	FUNCTION_BLOCK FB 141
	TITLE =G041M AERATION AIR STEEPING 5
	//COPYRIGHT:    (C) 2009  BUHLER AG, CH-9240 UZWIL, SWITZERLAND
	//
	//PRODUCT:      WinCoS_BIW01_09
	//
	//TITLE:        AERATION AIR STEEPING 5
	//                Machine group control
	//                Maschinengruppensteuerung
	//
	//--------------------------------------------------------------------------------
	//
	//IDENT:        AUTHOR:             DEPT:                              DATE:
	//
	//P01_FB141.1.0 K.Renz              CSB41                              13.Jan.2010
	//             1st Release
	//
	//--------------------------------------------------------------------------------
	//
	//PURPOSE:
	//
	//MANUAL :
	//
	//RESTRICTIONS:
	//
	//--------------------------------------------------------------------------------
	AUTHOR  : KR
	FAMILY  : USW
	VERSION : 9.9


	VAR
	  Gr       : FB10;	//Standard interface to group
	  InOutValue1    : DINT; //Data for user
	  InOutValue2    : DINT; //Data for user
	  OutWayConflict : BOOL;	//Data for user
	  OutSelectionOk : BOOL;	//Data for user
	  CmdNewValue : BOOL;	//Data for user
	  CmdNewJob   : BOOL;	//Data for user
	  OutCodeOK   : BOOL;	//Data for user
	  InEndOfJob  : BOOL ;	//Data for user
	  staWayOk      : BOOL ;	//Data for user
	  EdgeStartRelease : BOOL ;	//Data for user
	  USW8  : BOOL;	//Data for user
	  USW9 : BOOL;	//Data for user
	  USW10: BOOL;	//Data for user
	  USW11: BOOL;	//Data for user
	  USW12: BOOL;	//Data for user
	  USW13: BOOL;	//Data for user
	  USW14: BOOL;	//Data for user
	  USW15: BOOL;	//Data for user
	     #A_1115_QXV_BZS41_42 : FB13;   // VLS
	     #A_1115_MXZ45_BZS47_48 : FB13;   // VLS
	END_VAR
	VAR_TEMP
	   tmpEnable		: BOOL;
	   tmpFlag  		: BOOL;
	   tmpCmdNext		: BOOL;
	   tmpLocal  		: BOOL;
	   tmpAspOk  		: BOOL;
	   tmpHWStop 		: BOOL;
	   tmpInstanzDBNo       : INT ;
	END_VAR
	BEGIN
	NETWORK
	TITLE =
	NETWORK
	TITLE =Read command from group control
	//Parameter
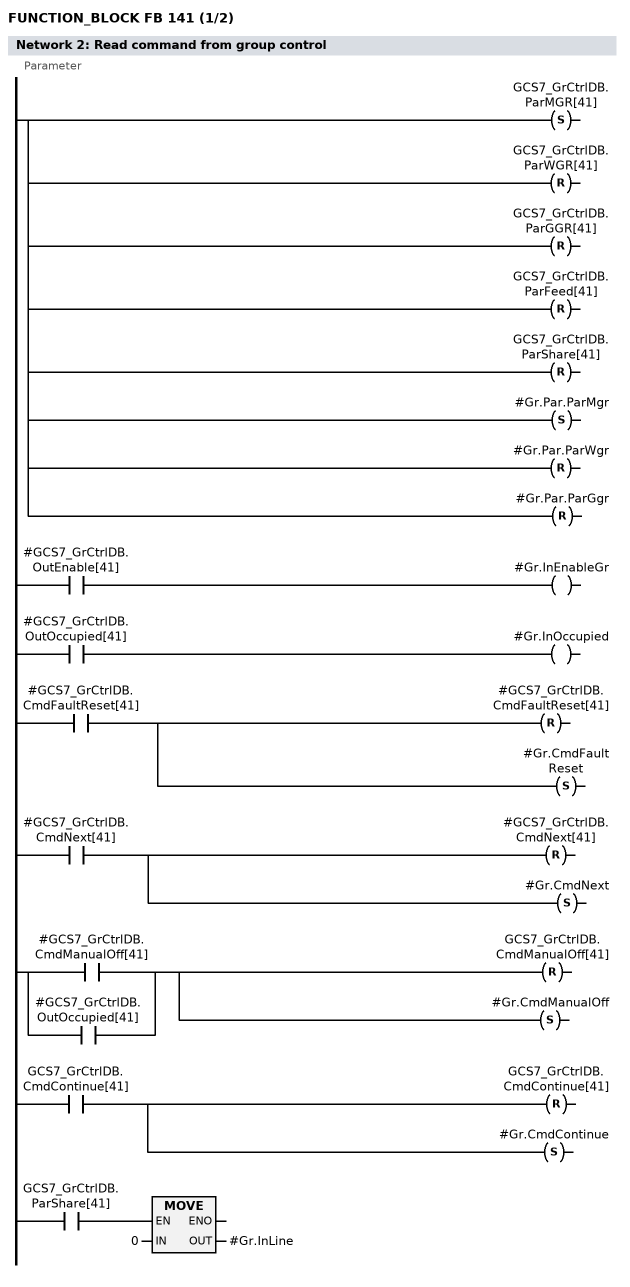
	      SET;
	      S   GCS7_GrCtrlDB.ParMGR[41];
	      R   GCS7_GrCtrlDB.ParWGR[41];
	      R   GCS7_GrCtrlDB.ParGGR[41];
	      R   GCS7_GrCtrlDB.ParFeed[41];
	      R   GCS7_GrCtrlDB.ParShare[41];
	      S   #Gr.Par.ParMgr;
	      R   #Gr.Par.ParWgr;
	      R   #Gr.Par.ParGgr;
	//Command
	      U   #GCS7_GrCtrlDB.OutEnable[41];
	      =   #Gr.InEnableGr;
	      U   #GCS7_GrCtrlDB.OutOccupied[41];
	      =   #Gr.InOccupied;
	      U   #GCS7_GrCtrlDB.CmdFaultReset[41];
	      R   #GCS7_GrCtrlDB.CmdFaultReset[41];
	      S   #Gr.CmdFaultReset;
	      U  #GCS7_GrCtrlDB.CmdNext[41];
	      R   #GCS7_GrCtrlDB.CmdNext[41];
	      S   #Gr.CmdNext;
	      U   #GCS7_GrCtrlDB.CmdManualOff[41];
	      O   #GCS7_GrCtrlDB.OutOccupied[41];
	      R   GCS7_GrCtrlDB.CmdManualOff[41];
	      S   #Gr.CmdManualOff;
	      U  GCS7_GrCtrlDB.CmdContinue[41];
	      R   GCS7_GrCtrlDB.CmdContinue[41];
	      S   #Gr.CmdContinue;
	//Init Line Number
	      U   GCS7_GrCtrlDB.ParShare[41];
	      SPBN WE00;
	      L     0;
	      T     #Gr.InLine;
	WE00: NOP   0;
	NETWORK
	TITLE =Call Methode Control
	// 1. Handle Interface PCControl
	// 2. Prepare mode --> ModePassive,ModeActive,ModeIdling
	// 3. Reset global flags of the group
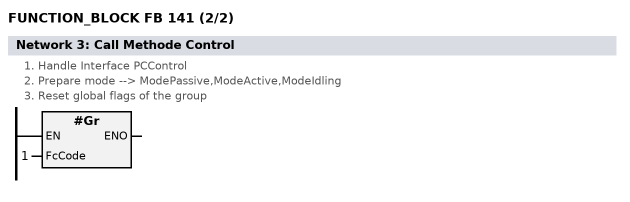
	      CALL #Gr (
	           FcCode                   := 1);
	NETWORK
	TITLE =Restart Idling Time
		L  #Gr.Par.ParIdling;
		L  2;
		>=I;
		SPB IdTm;
		T  #Gr.Par.ParIdling;
	IdTm:   NOP 0;
	      CLR;
	      S    #Gr.CmdRestartIdling;
	NETWORK
	TITLE =Prepare global flags
	NETWORK
	TITLE =Set Pattern (Target position)
	NETWORK
	TITLE =Interlocking WayOk
	//
	NETWORK
	TITLE =Interlocking Autostart
		CLR;
		R   #Gr.OutAutostart;
	NETWORK
	TITLE =Interlocking Enable
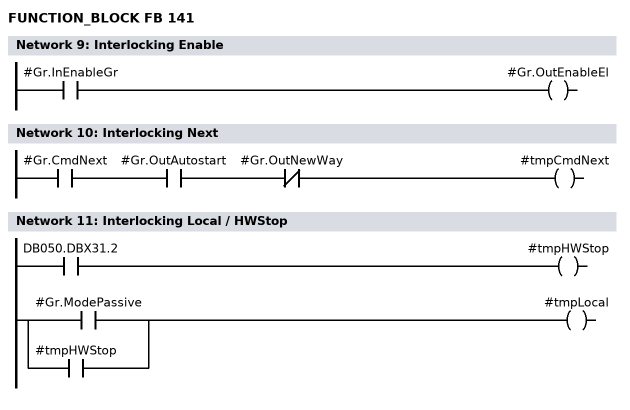
	      U     #Gr.InEnableGr;
	      =     #Gr.OutEnableEl;

	NETWORK
	TITLE =Interlocking Next
	      U     #Gr.CmdNext;
	      U     #Gr.OutAutostart;
	      UN    #Gr.OutNewWay;
	      =    #tmpCmdNext;

	NETWORK
	TITLE =Interlocking Local / HWStop
	      U    DB050.DBX31.2;
	      =    #tmpHWStop;

	      U    #Gr.ModePassive;
	      O    #tmpHWStop;
	      =    #tmpLocal;

	NETWORK
	TITLE =Interlocking Start Warning
	      NOP 0;
	//- Restart after fault --
	      U     #Gr.CmdFaultReset;
	      U     #Gr.VarFault;
	      S       "SYS_StartWarningDB".Area[1].CmdResetStartWarning;
	//- Run Timer --
	      AUF "G041M";
	      CALL  FB100 , DB100(
	       InModeHigher :=FALSE,
	       InArea     :=1,
	       InEnable   :=#Gr.OutEnableEl,
	       InLocal    :=#tmpLocal,
	       InStarted  :=#Gr.VarStarted,
	       InCmdNext  :=#tmpCmdNext,
	       OutCmdNext :=#tmpCmdNext,
	       OutStartwarning:=#Gr.VarStartWarning);
	//- Store Startwarning done  --
	//- Reset Autostart --
	      U     "SYS_StartWarningDB".TmpArea.OutStartReleaseRunningL;
	      FN    #EdgeStartRelease;
	      U     #Gr.VarFault;
	      R     #Gr.OutAutostart;
	NETWORK
	TITLE ==A-1115-QXV/BZS41/42 : AERATION AIR RING ST 5
	NOP 0;
	//-InLocal---
	      U     #tmpLocal;
	      =     #A_1115_QXV_BZS41_42.InLocal;
	//
	//-Interlocking---
	         =     #A_1115_QXV_BZS41_42.InEnableHN;
	         NOT;
	         =     #A_1115_QXV_BZS41_42.InEnableLN;
	//
	         SET;
	         S     #A_1115_QXV_BZS41_42.CmdNext;
	//
	      U     #Gr.OutSeqStop;
	      =     #A_1115_QXV_BZS41_42.InSeqStop;
	//
	//-Read inputs---
	      U     E 033.0;
	      =     #A_1115_QXV_BZS41_42.InpLN;
	      U     E 033.1;
	      =     #A_1115_QXV_BZS41_42.InpHN;
	      U   DB050.DBX31.2;
	      =     #A_1115_QXV_BZS41_42.InHWStop;
	       U     PLC_DPInfo.Master[1].SlavesError[6];
	       =       #A_1115_QXV_BZS41_42.InDPFault;
	//
	//-Set Parameters---
	//
	//-Call object control---
	      CALL  #A_1115_QXV_BZS41_42;
	//
	//-Write outputs---
	      U     #A_1115_QXV_BZS41_42.OutpHN;
	      =     A 033.1;
	NETWORK
	TITLE ==A-1115-MXZ45/BZS47/48 : AERATION AIR TUBE ST 5
	NOP 0;
	//-InLocal---
	      U     #tmpLocal;
	      =     #A_1115_MXZ45_BZS47_48.InLocal;
	//
	//-Interlocking---
	      	      U(;
	      U     #A_1115_QXV_BZS41_42.InEnableLN;
	      U     #A_1115_QXV_BZS41_42.StLN;
	      O;
	      U     #A_1115_QXV_BZS41_42.InEnableHN;
	      U     #A_1115_QXV_BZS41_42.StHN;
	      );
	         =     #A_1115_MXZ45_BZS47_48.InEnableHN;
	         NOT;
	         =     #A_1115_MXZ45_BZS47_48.InEnableLN;
	//
	         SET;
	         S     #A_1115_MXZ45_BZS47_48.CmdNext;
	//
	      U     #Gr.OutSeqStop;
	      =     #A_1115_MXZ45_BZS47_48.InSeqStop;
	//
	//-Read inputs---
	      U     E 066.2;
	      =     #A_1115_MXZ45_BZS47_48.InpLN;
	      U     E 066.3;
	      =     #A_1115_MXZ45_BZS47_48.InpHN;
	      X     A 065.1;
	      X     E 066.1;
	      O;
	      X     A 065.0;
	      X     E 066.0;
	      =     #A_1115_MXZ45_BZS47_48.InpFaultDev;
	      U   DB050.DBX31.2;
	      =     #A_1115_MXZ45_BZS47_48.InHWStop;
	       U     PLC_DPInfo.Master[1].SlavesError[10];
	       =       #A_1115_MXZ45_BZS47_48.InDPFault;
	//
	//-Set Parameters---
	//
	//-Call object control---
	      CALL  #A_1115_MXZ45_BZS47_48;
	//
	//-Write outputs---
	      U     #A_1115_MXZ45_BZS47_48.OutpLN;
	      =     A 065.1;
	      U     #A_1115_MXZ45_BZS47_48.OutpHN;
	      =     A 065.0;
	NETWORK
	TITLE =Test Fault
	      U     #A_1115_QXV_BZS41_42.StFault;
	      O     #A_1115_MXZ45_BZS47_48.StFault;
	      =     #Gr.VarFault;
	NETWORK
	TITLE =Test Warning
	      CLR;
	      =     #Gr.OutWarning;
	NETWORK
	TITLE =Test Stopped
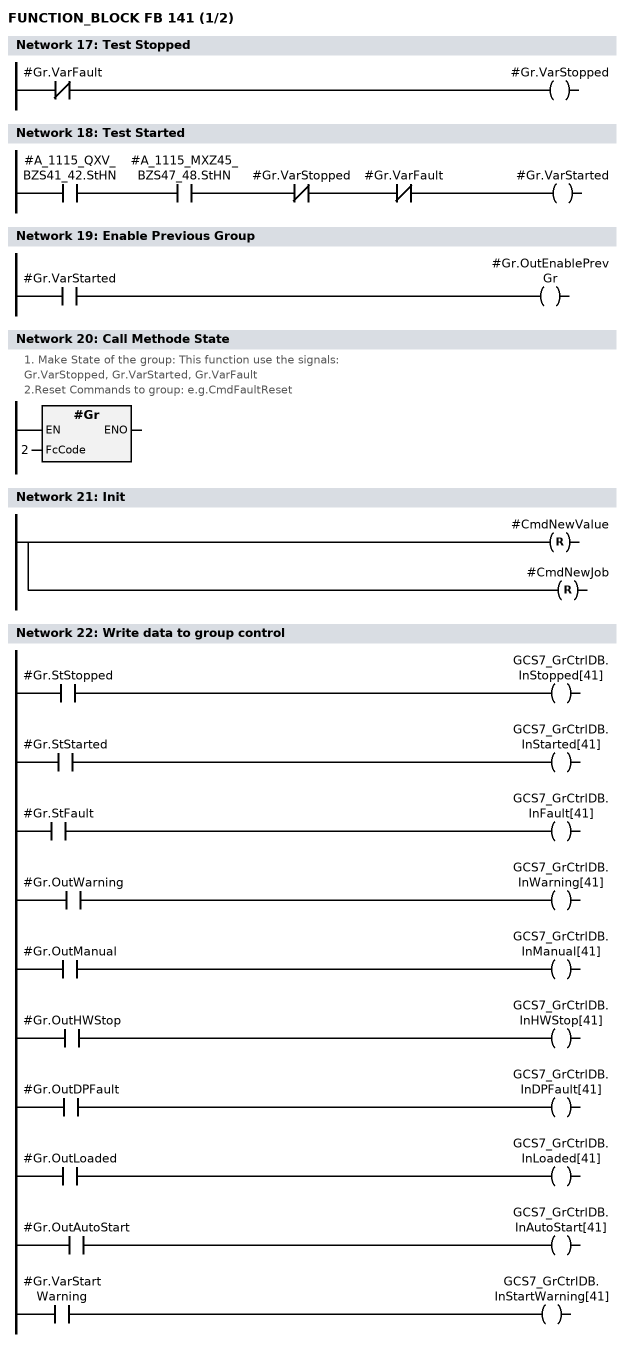
	      UN   #Gr.VarFault;
	      =     #Gr.VarStopped;
	NETWORK
	TITLE =Test Started
	      U     #A_1115_QXV_BZS41_42.StHN;
	      U     #A_1115_MXZ45_BZS47_48.StHN;
	      UN  #Gr.VarStopped;
	      UN  #Gr.VarFault;
	      =     #Gr.VarStarted;
	NETWORK
	TITLE =Enable Previous Group
	      U    #Gr.VarStarted;
	      =     #Gr.OutEnablePrevGr;
	NETWORK
	TITLE =Call Methode State
	//1. Make State of the group: This function use the signals:
	//        Gr.VarStopped, Gr.VarStarted, Gr.VarFault
	//2.Reset Commands to group: e.g.CmdFaultReset
	      CALL #Gr (
	           FcCode                   := 2);
	NETWORK
	TITLE =Init
	      SET;
	      R    #CmdNewValue;
	      R    #CmdNewJob;
	NETWORK
	TITLE =Write data to group control
	      U   #Gr.StStopped;
	      =   GCS7_GrCtrlDB.InStopped[41];
	      U   #Gr.StStarted;
	      =   GCS7_GrCtrlDB.InStarted[41];
	      U   #Gr.StFault;
	      =   GCS7_GrCtrlDB.InFault[41];
	      U   #Gr.OutWarning;
	      =   GCS7_GrCtrlDB.InWarning[41];
	      U   #Gr.OutManual;
	      =   GCS7_GrCtrlDB.InManual[41];
	      U   #Gr.OutHWStop;
	      =   GCS7_GrCtrlDB.InHWStop[41];
	      U   #Gr.OutDPFault;
	      =   GCS7_GrCtrlDB.InDPFault[41];
	      U   #Gr.OutLoaded;
	      =   GCS7_GrCtrlDB.InLoaded[41];
	      U   #Gr.OutAutoStart;
	      =   GCS7_GrCtrlDB.InAutoStart[41];
	      U   #Gr.VarStartWarning;
	      =   GCS7_GrCtrlDB.InStartWarning[41];
	NETWORK
	TITLE =End of block
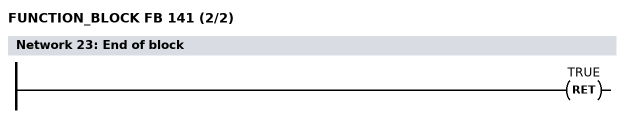

	BE

	END_FUNCTION_BLOCK
